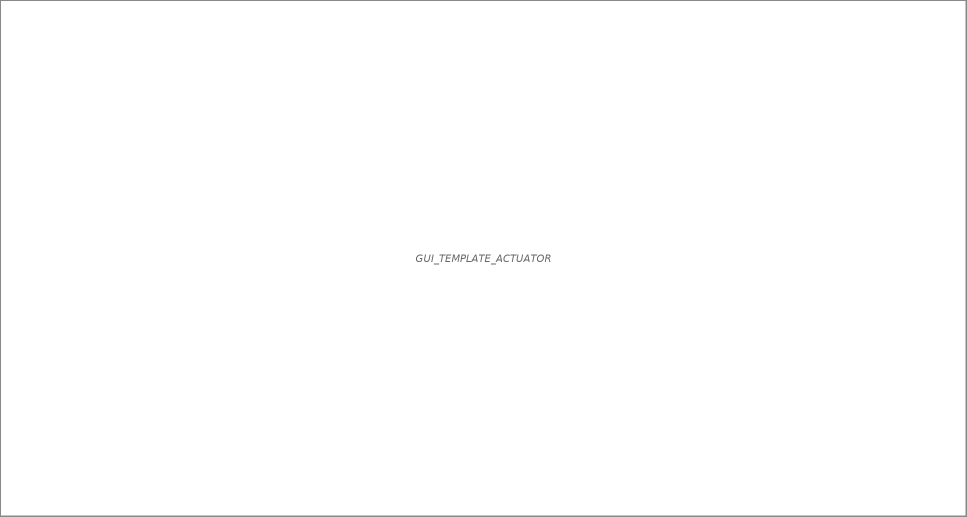
VISUALIZATION GUI_Actuator004  // 967x517
    Frame (0,0 967x517)
        shows GUI_TEMPLATE_ACTUATOR(m_Instance := MAIN.Actuator004)
END_VISUALIZATION

(* stored: Version 1.1.0.1, ProductVersion 3.1.4024.3
   Visu GUI_Actuator004: Id {f2206a03-2239-4bb4-8bde-0da694a6053b} *)
